PROGRAM PRG_House
VAR
	hall : Hall;
END_VAR


	hall();
	

////	IO Mapping:
////	Hall:
//	EL1008_01;
//	EL1008_02;
//	EL1008_03;
//	EL2008_01;
//	EL2008_02;
//	EL4004_01;
	
////	Kitchen
//	EL1008_04;
//	EL2008_03;
//	EL4004_02;
	
////	Bedroom1
//	EL1008_05;
//	EL1008_06;
//	EL2008_04;
//	EL4004_03;
	
////	Bedroom2
//	EL1008_07;
//	EL1008_08;
//	EL2008_05;
//	EL4004_04;

END_PROGRAM

(* stored: Version 1.1.0.1, ProductVersion 3.1.4024.13
   POU PRG_House: Id {de77fefd-9b7f-419a-b0ed-9b272890e3cb}, SpecialFunc None *)
